// TIA Portal V19 export
FUNCTION_BLOCK "CallUnit"   // FB130, LAD
TITLE = CallUnit
AUTHOR : Siemens_FA_SUP
// This block calls all functionality inside the unit.
// stored: IsIECCheckEnabled true, MemoryReserve 100, Namespace Unit, SetENOAutomatically true
   VAR_INPUT
      safetyReleased : Bool;   // Status from safety program
   END_VAR
   VAR_OUTPUT
      acknowledgeSafety { ExternalWritable := 'False'} : Bool;   // Acknowledge command to the safety program
   END_VAR
   VAR_IN_OUT
      globalStatus : "LAF_typeGeneralStatus";   // Global status
      unitInterface : "LAF_typeUnitInterface";   // Global unit interface
   END_VAR
   VAR
      statRemoteInterface { ExternalWritable := 'False'} : "LUC_typeCommands";
      instManageAlarms { ExternalWritable := 'False'} : "LAF_ManageAlarms";
      instStatusCollector { ExternalWritable := 'False'} : "LUC_StatusCollector";
      instInterfaceManager { ExternalWritable := 'False'} : "LUC_InterfaceManager";
      instUnitModeStateManager { ExternalWritable := 'False'} : "LPMLV2022_UnitModeStateManager";
      instRemoteInterfaceOpcUa { ExternalWritable := 'False'} : "LUC_RemoteCtrl_OpcUa";
      instSignalStack { ExternalWritable := 'False'} : "LUC_SignalStack";
      instUnitModeStateTimes { ExternalWritable := 'False'} : "LPMLV2022_UnitModeStateTimes";
      instUnitModeChangeAllowed { ExternalWritable := 'False'} : "LPMLV2022_UnitModeChangeAllowed";
   END_VAR
   VAR_TEMP
      tempUnitFeedback : "LUC_typeStateCommands";   // Collected commands in the unit, e.g. direct command or commands derived from alarms
      tempProcessCommands : "LUC_typeStateCommands";   // Requested unit state changes by the process
      tempUnitMode : DInt;   // Requested unit mode
      tempUnitModeChangeRequest : Bool;   // Request unit mode
      tempCntrlCmd : DInt;   // Request control command
      tempCmdChangeRequest : Bool;   // Enable change into requested state
      tempSc : Bool;   // State change from FALSE to TRUE (rising edge) triggers state complete signal
   END_VAR
BEGIN

REGION Network 1: BLOCK INFO HEADER
   // (company) / (C) Copyright (year)
   // ---------------------------------------------------------------------------------
   // Title:                             (Title of this block)
   // Comment/Function: (that is implemented in the block)
   // Library/Family:           (that the source is dedicated to)
   // Author:                        (department / person in charge / contact)
   // Target System:          (test system with FW version)
   // Engineering:              TIA Portal (SW version)
   // Restrictions:               (OB types, etc.)
   // Requirements:           (hardware, technological package, etc.)
   // ---------------------------------------------------------------------------------
   // Change log table:
   // Version          | Date             | Signature      | Expert in charge  | Changes applied ------------------------|----------------------|-------------------------|--------------------------------|-----------------------
   // 001.000.000 | yyyy-mm-dd | 0x00000000 | (name of expert) | First released version
END_REGION

REGION Network 2: DESCRIPTION
   // This is a template block provided by the Automation Framework. It can be used to create an own project.
   // The Block Info Header is prepared to put in your own data.
   // Description of the block could be added here and the docu created by Code2Docu.
END_REGION

REGION Network 3: Simulation
   // If simulation is active on a global level, inherit this status and set simulation active in this unit also. Information is written to DB ControlNodes, from where it is distributed to the equipmemt modules.
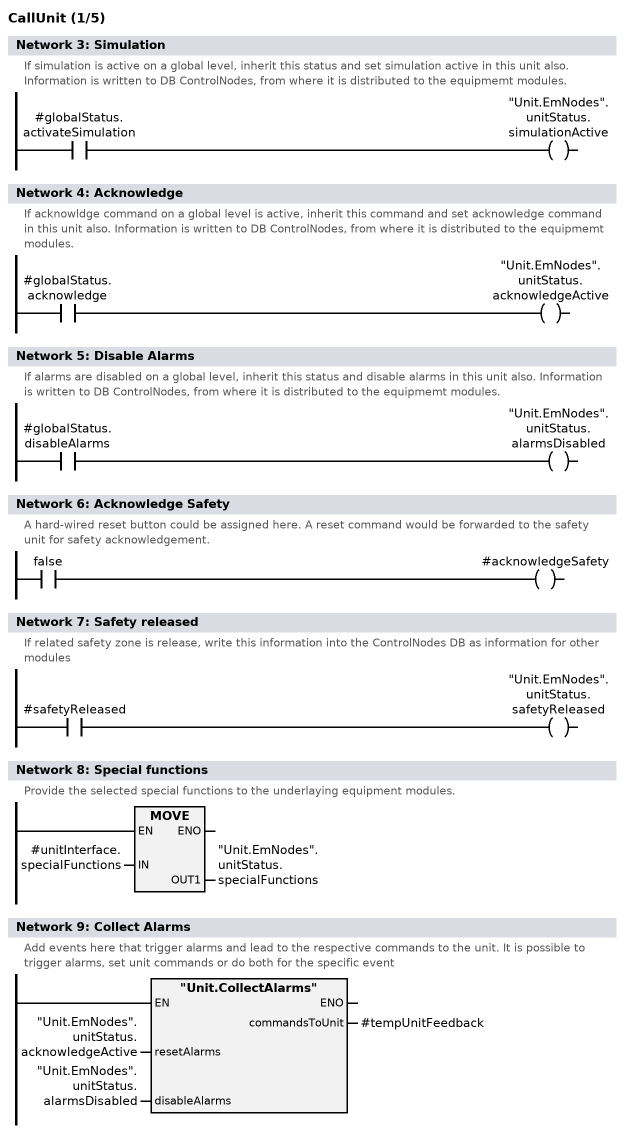
   RUNG wire#powerrail
      Contact( #globalStatus.activateSimulation )
      Coil( "Unit.EmNodes".unitStatus.simulationActive )
   END_RUNG
   // the same network as SCL:
   "Unit.EmNodes".unitStatus.simulationActive := #globalStatus.activateSimulation;
END_REGION

REGION Network 4: Acknowledge
   // If acknowldge command on a global level is active, inherit this command and set acknowledge command in this unit also. Information is written to DB ControlNodes, from where it is distributed to the equipmemt modules.
   RUNG wire#powerrail
      Contact( #globalStatus.acknowledge )
      Coil( "Unit.EmNodes".unitStatus.acknowledgeActive )
   END_RUNG
   // the same network as SCL:
   "Unit.EmNodes".unitStatus.acknowledgeActive := #globalStatus.acknowledge;
END_REGION

REGION Network 5: Disable Alarms
   // If alarms are disabled on a global level, inherit this status and disable alarms in this unit also. Information is written to DB ControlNodes, from where it is distributed to the equipmemt modules.
   RUNG wire#powerrail
      Contact( #globalStatus.disableAlarms )
      Coil( "Unit.EmNodes".unitStatus.alarmsDisabled )
   END_RUNG
   // the same network as SCL:
   "Unit.EmNodes".unitStatus.alarmsDisabled := #globalStatus.disableAlarms;
END_REGION

REGION Network 6: Acknowledge Safety
   // A hard-wired reset button could be assigned here. A reset command would be forwarded to the safety unit for safety acknowledgement.
   RUNG wire#powerrail
      Contact( false )
      Coil( #acknowledgeSafety )
   END_RUNG
   // the same network as SCL:
   #acknowledgeSafety := false;
END_REGION

REGION Network 7: Safety released
   // If related safety zone is release, write this information into the ControlNodes DB as information for other modules
   RUNG wire#powerrail
      Contact( #safetyReleased )
      Coil( "Unit.EmNodes".unitStatus.safetyReleased )
   END_RUNG
   // the same network as SCL:
   "Unit.EmNodes".unitStatus.safetyReleased := #safetyReleased;
END_REGION

REGION Network 8: Special functions
   // Provide the selected special functions to the underlaying equipment modules.
   RUNG wire#powerrail
      Move(in := #unitInterface.specialFunctions, out1 => "Unit.EmNodes".unitStatus.specialFunctions)
   END_RUNG
   // the same network as SCL:
   "Unit.EmNodes".unitStatus.specialFunctions := #unitInterface.specialFunctions;
END_REGION

REGION Network 9: Collect Alarms
   // Add events here that trigger alarms and lead to the respective commands to the unit. It is possible to trigger alarms, set unit commands or do both for the specific event
   RUNG wire#powerrail
      "Unit.CollectAlarms"(resetAlarms := "Unit.EmNodes".unitStatus.acknowledgeActive, disableAlarms := "Unit.EmNodes".unitStatus.alarmsDisabled, commandsToUnit => #tempUnitFeedback)
   END_RUNG
   // the same network as SCL:
   "Unit.CollectAlarms"(resetAlarms := "Unit.EmNodes".unitStatus.acknowledgeActive,
                        disableAlarms := "Unit.EmNodes".unitStatus.alarmsDisabled,
                        commandsToUnit => #tempUnitFeedback);
END_REGION

REGION Network 10: Manage Alarms
   // Derive commands from the ProDiag supervision. The ProDiag supervisions contain categories which define the reaction of these supervisions (e.g. abort, stop, hold). These are handed over as commands to the unit level.
   // Alternatively, if no ProDiag should be used, you can use the LAF_ManageBitAlarms to realize bit alarm handling. This block can be found in LAF in folder 70_AlarmHandling.
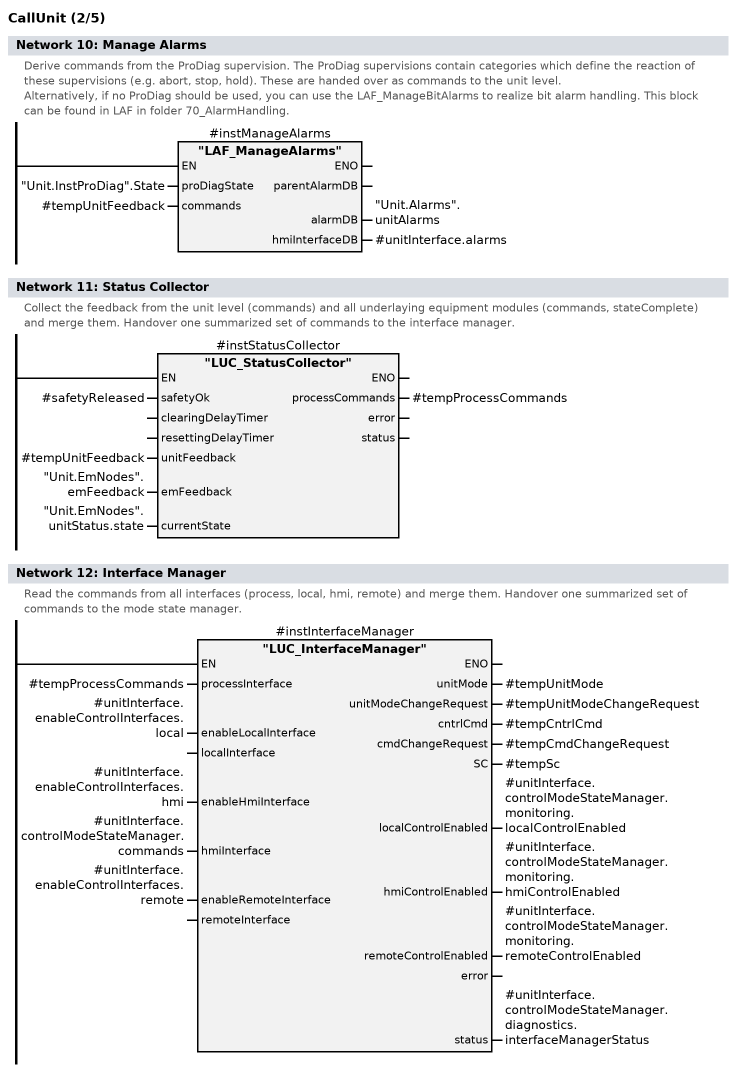
   RUNG wire#powerrail
      #instManageAlarms(proDiagState := "Unit.InstProDiag".State, commands := #tempUnitFeedback, parentAlarmDB =>, alarmDB => "Unit.Alarms".unitAlarms, hmiInterfaceDB => #unitInterface.alarms)
   END_RUNG
   // the same network as SCL:
   #instManageAlarms(proDiagState := "Unit.InstProDiag".State,   // "LAF_ManageAlarms"
                     commands := #tempUnitFeedback,
                     alarmDB => "Unit.Alarms".unitAlarms,
                     hmiInterfaceDB => #unitInterface.alarms);
END_REGION

REGION Network 11: Status Collector
   // Collect the feedback from the unit level (commands) and all underlaying equipment modules (commands, stateComplete) and merge them. Handover one summarized set of commands to the interface manager.
   RUNG wire#powerrail
      #instStatusCollector(safetyOk := #safetyReleased, clearingDelayTimer :=, resettingDelayTimer :=, unitFeedback := #tempUnitFeedback, emFeedback := "Unit.EmNodes".emFeedback, currentState := "Unit.EmNodes".unitStatus.state, processCommands => #tempProcessCommands, error =>, status =>)
   END_RUNG
   // the same network as SCL:
   #instStatusCollector(safetyOk := #safetyReleased,   // "LUC_StatusCollector"
                        unitFeedback := #tempUnitFeedback,
                        emFeedback := "Unit.EmNodes".emFeedback,
                        currentState := "Unit.EmNodes".unitStatus.state,
                        processCommands => #tempProcessCommands);
END_REGION

REGION Network 12: Interface Manager
   // Read the commands from all interfaces (process, local, hmi, remote) and merge them. Handover one summarized set of commands to the mode state manager.
   RUNG wire#powerrail
      #instInterfaceManager(processInterface := #tempProcessCommands, enableLocalInterface := #unitInterface.enableControlInterfaces.local, localInterface :=, enableHmiInterface := #unitInterface.enableControlInterfaces.hmi, hmiInterface := #unitInterface.controlModeStateManager.commands, enableRemoteInterface := #unitInterface.enableControlInterfaces.remote, remoteInterface :=, unitMode => #tempUnitMode, unitModeChangeRequest => #tempUnitModeChangeRequest, cntrlCmd => #tempCntrlCmd, cmdChangeRequest => #tempCmdChangeRequest, SC => #tempSc, localControlEnabled => #unitInterface.controlModeStateManager.monitoring.localControlEnabled, hmiControlEnabled => #unitInterface.controlModeStateManager.monitoring.hmiControlEnabled, remoteControlEnabled => #unitInterface.controlModeStateManager.monitoring.remoteControlEnabled, error =>, status => #unitInterface.controlModeStateManager.diagnostics.interfaceManagerStatus)
   END_RUNG
   // the same network as SCL:
   #instInterfaceManager(processInterface := #tempProcessCommands,   // "LUC_InterfaceManager"
                         enableLocalInterface := #unitInterface.enableControlInterfaces.local,
                         enableHmiInterface := #unitInterface.enableControlInterfaces.hmi,
                         hmiInterface := #unitInterface.controlModeStateManager.commands,
                         enableRemoteInterface := #unitInterface.enableControlInterfaces.remote,
                         unitMode => #tempUnitMode,
                         unitModeChangeRequest => #tempUnitModeChangeRequest,
                         cntrlCmd => #tempCntrlCmd,
                         cmdChangeRequest => #tempCmdChangeRequest,
                         SC => #tempSc,
                         localControlEnabled => #unitInterface.controlModeStateManager.monitoring.localControlEnabled,
                         hmiControlEnabled => #unitInterface.controlModeStateManager.monitoring.hmiControlEnabled,
                         remoteControlEnabled => #unitInterface.controlModeStateManager.monitoring.remoteControlEnabled,
                         status => #unitInterface.controlModeStateManager.diagnostics.interfaceManagerStatus);
END_REGION

REGION Network 13: Mode and State Manager
   // Determine unit mode and state based on the collected commands and status
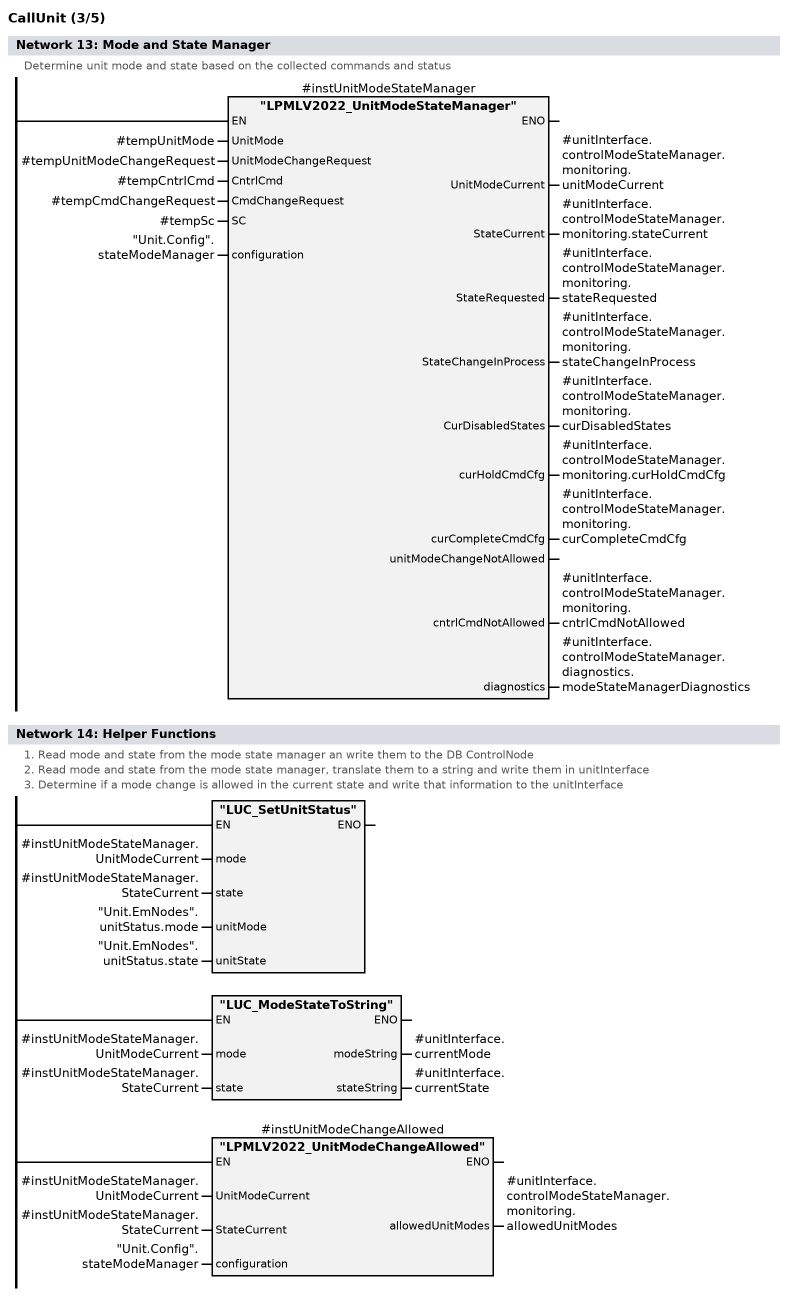
   RUNG wire#powerrail
      #instUnitModeStateManager(UnitMode := #tempUnitMode, UnitModeChangeRequest := #tempUnitModeChangeRequest, CntrlCmd := #tempCntrlCmd, CmdChangeRequest := #tempCmdChangeRequest, SC := #tempSc, configuration := "Unit.Config".stateModeManager, UnitModeCurrent => #unitInterface.controlModeStateManager.monitoring.unitModeCurrent, StateCurrent => #unitInterface.controlModeStateManager.monitoring.stateCurrent, StateRequested => #unitInterface.controlModeStateManager.monitoring.stateRequested, StateChangeInProcess => #unitInterface.controlModeStateManager.monitoring.stateChangeInProcess, CurDisabledStates => #unitInterface.controlModeStateManager.monitoring.curDisabledStates, curHoldCmdCfg => #unitInterface.controlModeStateManager.monitoring.curHoldCmdCfg, curCompleteCmdCfg => #unitInterface.controlModeStateManager.monitoring.curCompleteCmdCfg, unitModeChangeNotAllowed =>, cntrlCmdNotAllowed => #unitInterface.controlModeStateManager.monitoring.cntrlCmdNotAllowed, diagnostics => #unitInterface.controlModeStateManager.diagnostics.modeStateManagerDiagnostics)
   END_RUNG
   // the same network as SCL:
   #instUnitModeStateManager(UnitMode := #tempUnitMode,   // "LPMLV2022_UnitModeStateManager"
                           UnitModeChangeRequest := #tempUnitModeChangeRequest,
                           CntrlCmd := #tempCntrlCmd,
                           CmdChangeRequest := #tempCmdChangeRequest,
                           SC := #tempSc,
                           configuration := "Unit.Config".stateModeManager,
                           UnitModeCurrent => #unitInterface.controlModeStateManager.monitoring.unitModeCurrent,
                           StateCurrent => #unitInterface.controlModeStateManager.monitoring.stateCurrent,
                           StateRequested => #unitInterface.controlModeStateManager.monitoring.stateRequested,
                           StateChangeInProcess => #unitInterface.controlModeStateManager.monitoring.stateChangeInProcess,
                           CurDisabledStates => #unitInterface.controlModeStateManager.monitoring.curDisabledStates,
                           curHoldCmdCfg => #unitInterface.controlModeStateManager.monitoring.curHoldCmdCfg,
                           curCompleteCmdCfg => #unitInterface.controlModeStateManager.monitoring.curCompleteCmdCfg,
                           cntrlCmdNotAllowed => #unitInterface.controlModeStateManager.monitoring.cntrlCmdNotAllowed,
                           diagnostics => #unitInterface.controlModeStateManager.diagnostics.modeStateManagerDiagnostics);
END_REGION

REGION Network 14: Helper Functions
   // 1. Read mode and state from the mode state manager an write them to the DB ControlNode
   // 2. Read mode and state from the mode state manager, translate them to a string and write them in unitInterface
   // 3. Determine if a mode change is allowed in the current state and write that information to the unitInterface
   RUNG wire#powerrail
      "LUC_SetUnitStatus"(mode := #instUnitModeStateManager.UnitModeCurrent, state := #instUnitModeStateManager.StateCurrent, unitMode := "Unit.EmNodes".unitStatus.mode, unitState := "Unit.EmNodes".unitStatus.state)
   END_RUNG
   RUNG wire#powerrail
      "LUC_ModeStateToString"(mode := #instUnitModeStateManager.UnitModeCurrent, state := #instUnitModeStateManager.StateCurrent, modeString => #unitInterface.currentMode, stateString => #unitInterface.currentState)
   END_RUNG
   RUNG wire#powerrail
      #instUnitModeChangeAllowed(UnitModeCurrent := #instUnitModeStateManager.UnitModeCurrent, StateCurrent := #instUnitModeStateManager.StateCurrent, configuration := "Unit.Config".stateModeManager, allowedUnitModes => #unitInterface.controlModeStateManager.monitoring.allowedUnitModes)
   END_RUNG
   // the same network as SCL:
   "LUC_SetUnitStatus"(mode := #instUnitModeStateManager.UnitModeCurrent,
                       state := #instUnitModeStateManager.StateCurrent,
                       unitMode := "Unit.EmNodes".unitStatus.mode,
                       unitState := "Unit.EmNodes".unitStatus.state);
   "LUC_ModeStateToString"(mode := #instUnitModeStateManager.UnitModeCurrent,
                           state := #instUnitModeStateManager.StateCurrent,
                           modeString => #unitInterface.currentMode,
                           stateString => #unitInterface.currentState);
   #instUnitModeChangeAllowed(UnitModeCurrent := #instUnitModeStateManager.UnitModeCurrent,   // "LPMLV2022_UnitModeChangeAllowed"
                           StateCurrent := #instUnitModeStateManager.StateCurrent,
                           configuration := "Unit.Config".stateModeManager,
                           allowedUnitModes => #unitInterface.controlModeStateManager.monitoring.allowedUnitModes);
END_REGION

REGION Network 15: History
   // Update the mode and state history. When mode or state change occur, save current mode and state in history[0] and the previous ones in ascending order.
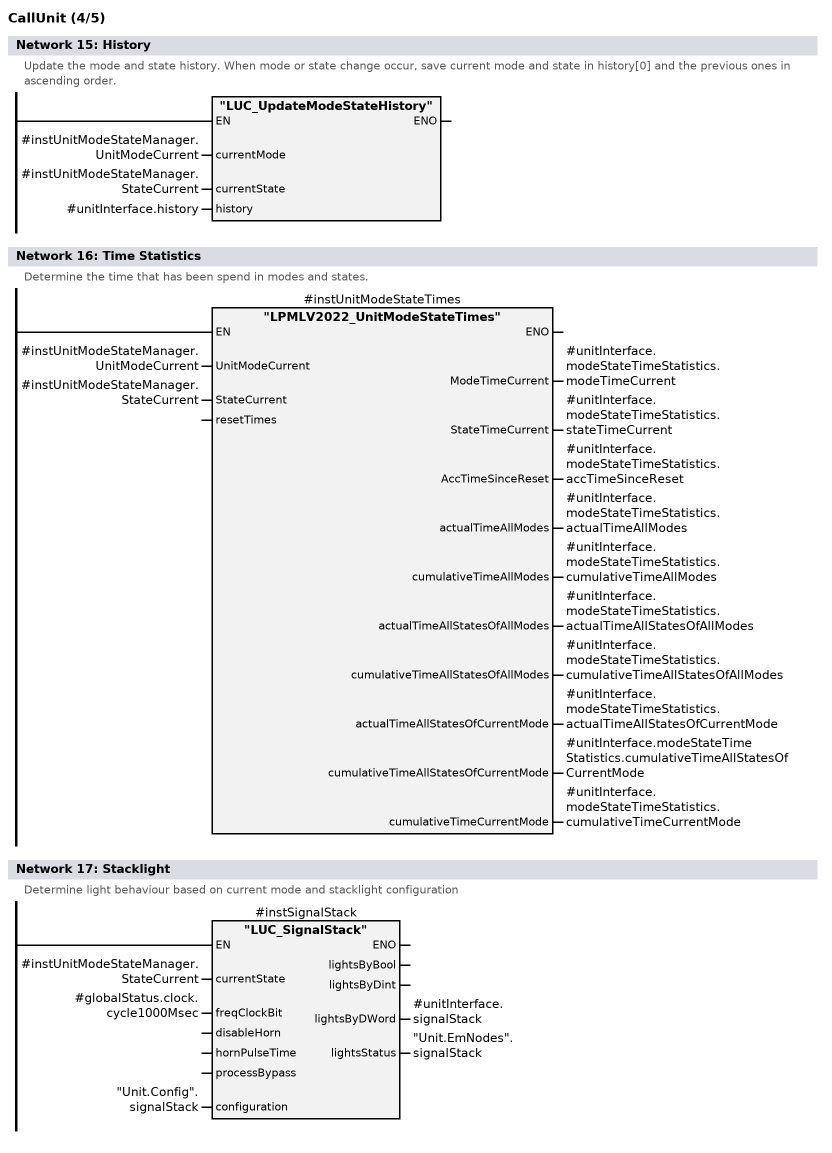
   RUNG wire#powerrail
      "LUC_UpdateModeStateHistory"(currentMode := #instUnitModeStateManager.UnitModeCurrent, currentState := #instUnitModeStateManager.StateCurrent, history := #unitInterface.history)
   END_RUNG
   // the same network as SCL:
   "LUC_UpdateModeStateHistory"(currentMode := #instUnitModeStateManager.UnitModeCurrent,
                           currentState := #instUnitModeStateManager.StateCurrent,
                           history := #unitInterface.history);
END_REGION

REGION Network 16: Time Statistics
   // Determine the time that has been spend in modes and states.
   RUNG wire#powerrail
      #instUnitModeStateTimes(UnitModeCurrent := #instUnitModeStateManager.UnitModeCurrent, StateCurrent := #instUnitModeStateManager.StateCurrent, resetTimes :=, ModeTimeCurrent => #unitInterface.modeStateTimeStatistics.modeTimeCurrent, StateTimeCurrent => #unitInterface.modeStateTimeStatistics.stateTimeCurrent, AccTimeSinceReset => #unitInterface.modeStateTimeStatistics.accTimeSinceReset, actualTimeAllModes => #unitInterface.modeStateTimeStatistics.actualTimeAllModes, cumulativeTimeAllModes => #unitInterface.modeStateTimeStatistics.cumulativeTimeAllModes, actualTimeAllStatesOfAllModes => #unitInterface.modeStateTimeStatistics.actualTimeAllStatesOfAllModes, cumulativeTimeAllStatesOfAllModes => #unitInterface.modeStateTimeStatistics.cumulativeTimeAllStatesOfAllModes, actualTimeAllStatesOfCurrentMode => #unitInterface.modeStateTimeStatistics.actualTimeAllStatesOfCurrentMode, cumulativeTimeAllStatesOfCurrentMode => #unitInterface.modeStateTimeStatistics.cumulativeTimeAllStatesOfCurrentMode, cumulativeTimeCurrentMode => #unitInterface.modeStateTimeStatistics.cumulativeTimeCurrentMode)
   END_RUNG
   // the same network as SCL:
   #instUnitModeStateTimes(UnitModeCurrent := #instUnitModeStateManager.UnitModeCurrent,   // "LPMLV2022_UnitModeStateTimes"
                           StateCurrent := #instUnitModeStateManager.StateCurrent,
                           ModeTimeCurrent => #unitInterface.modeStateTimeStatistics.modeTimeCurrent,
                           StateTimeCurrent => #unitInterface.modeStateTimeStatistics.stateTimeCurrent,
                           AccTimeSinceReset => #unitInterface.modeStateTimeStatistics.accTimeSinceReset,
                           actualTimeAllModes => #unitInterface.modeStateTimeStatistics.actualTimeAllModes,
                           cumulativeTimeAllModes => #unitInterface.modeStateTimeStatistics.cumulativeTimeAllModes,
                           actualTimeAllStatesOfAllModes => #unitInterface.modeStateTimeStatistics.actualTimeAllStatesOfAllModes,
                           cumulativeTimeAllStatesOfAllModes => #unitInterface.modeStateTimeStatistics.cumulativeTimeAllStatesOfAllModes,
                           actualTimeAllStatesOfCurrentMode => #unitInterface.modeStateTimeStatistics.actualTimeAllStatesOfCurrentMode,
                           cumulativeTimeAllStatesOfCurrentMode => #unitInterface.modeStateTimeStatistics.cumulativeTimeAllStatesOfCurrentMode,
                           cumulativeTimeCurrentMode => #unitInterface.modeStateTimeStatistics.cumulativeTimeCurrentMode);
END_REGION

REGION Network 17: Stacklight
   // Determine light behaviour based on current mode and stacklight configuration
   RUNG wire#powerrail
      #instSignalStack(currentState := #instUnitModeStateManager.StateCurrent, freqClockBit := #globalStatus.clock.cycle1000Msec, disableHorn :=, hornPulseTime :=, processBypass :=, configuration := "Unit.Config".signalStack, lightsByBool =>, lightsByDint =>, lightsByDWord => #unitInterface.signalStack, lightsStatus => "Unit.EmNodes".signalStack)
   END_RUNG
   // the same network as SCL:
   #instSignalStack(currentState := #instUnitModeStateManager.StateCurrent,   // "LUC_SignalStack"
                    freqClockBit := #globalStatus.clock.cycle1000Msec,
                    configuration := "Unit.Config".signalStack,
                    lightsByDWord => #unitInterface.signalStack,
                    lightsStatus => "Unit.EmNodes".signalStack);
END_REGION

REGION Network 18: Remote Control via OPC UA
   // Control the mode state manager remotely via OPC UA
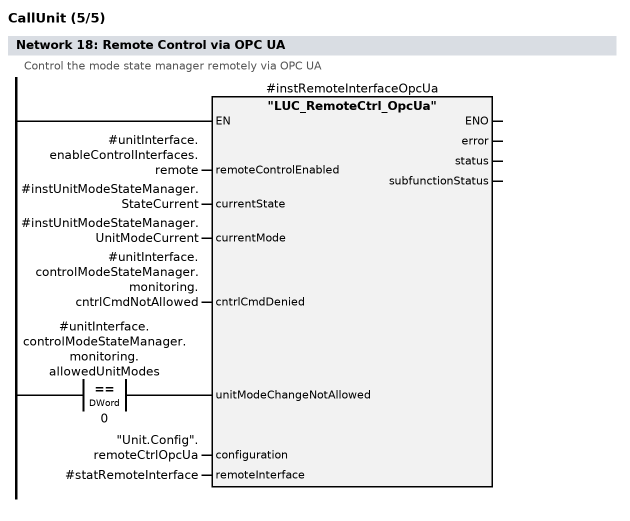
   RUNG wire#powerrail
      #instRemoteInterfaceOpcUa(unitModeChangeNotAllowed := wire#w1, remoteControlEnabled := #unitInterface.enableControlInterfaces.remote, currentState := #instUnitModeStateManager.StateCurrent, currentMode := #instUnitModeStateManager.UnitModeCurrent, cntrlCmdDenied := #unitInterface.controlModeStateManager.monitoring.cntrlCmdNotAllowed, configuration := "Unit.Config".remoteCtrlOpcUa, remoteInterface := #statRemoteInterface, error =>, status =>, subfunctionStatus =>)
   END_RUNG
   RUNG wire#powerrail
      { S7_Templates := "SrcType := DWord" } EQ_Contact(in1 := #unitInterface.controlModeStateManager.monitoring.allowedUnitModes, in2 := 0)
   END_RUNG wire#w1
   // the same network as SCL:
   #instRemoteInterfaceOpcUa(remoteControlEnabled := #unitInterface.enableControlInterfaces.remote,   // "LUC_RemoteCtrl_OpcUa"
                           currentState := #instUnitModeStateManager.StateCurrent,
                           currentMode := #instUnitModeStateManager.UnitModeCurrent,
                           cntrlCmdDenied := #unitInterface.controlModeStateManager.monitoring.cntrlCmdNotAllowed,
                           unitModeChangeNotAllowed := #unitInterface.controlModeStateManager.monitoring.allowedUnitModes = 0,
                           configuration := "Unit.Config".remoteCtrlOpcUa,
                           remoteInterface := #statRemoteInterface);
END_REGION
END_FUNCTION_BLOCK
